// TIA Portal V20 export
VAR_GLOBAL   // PLC tag table "Default tag table"
   Tag_1 AT %M10.0 : Bool;
   Tag_2 AT %M10.1 : Bool;
END_VAR
